FUNCTION_BLOCK L1_ControllerBase_SFC

VAR CONSTANT
	MAX_ERRORS	: UINT := 10;
	MAX_TIMEOUT	: TIME := T#30S;
END_VAR

VAR_INPUT
	dr			: REFERENCE TO L1_Director;		// acceso a todos los tiempos de espera
	IC			: BOOL;
	Execute		: BOOL;
	Ack			: BOOL;	
	SFCPause	: BOOL;
	SFCReset	: BOOL;
	UnsafeStop 	: BOOL := FALSE;
	Clocks		: ARRAY[1..MAX_ERRORS]	OF TON; 
END_VAR

VAR_OUTPUT
	Ready		: BOOL;
	Done		: BOOL := FALSE;
	Timed		: ARRAY[1..MAX_ERRORS]	OF BOOL; 
	NumError	: UINT := 0;
	gmModePrev	: L1_GEMMA := L1_GEMMA.A6Inicializando;
	
	colPicFill	: DWORD; // color para destacar en la foto según esté Ready (tranparente), Ejecutando (amarillo) o Esperando Ack (verde) 
	colPicFram	: DWORD; // color del marco  	
END_VAR

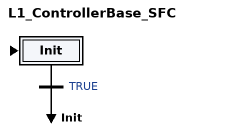
INITIAL_STEP Init:
END_STEP
TRANSITION FROM Init TO Init
    := TRUE;
END_TRANSITION

METHOD FB_init : BOOL
VAR_INPUT
	bInitRetains : BOOL; // if TRUE, the retain variables are initialized (warm start / cold start)
	bInCopyCode : BOOL;  // if TRUE, the instance afterwards gets moved into the copy code (online change)
END_VAR

VAR 
	I: UINT;
END_VAR
NumError		:= 0;					// Inicializar el estado a 0 (no hay error)

FOR I:=1 TO MAX_ERRORS DO				// Inicializar todos los flags de etapas temporizadas
	Timed[i] 		:= FALSE;
	//Clocks[i].IN	:= Timed[i];
	//Clocks[i].PT	:= MAX_TIMEOUT;	
END_FOR
END_METHOD

METHOD IsPaused : BOOL
IsPaused := SFCPause;
END_METHOD

METHOD ProcessCycle : BOOL

VAR_INPUT
	gmMode : L1_GEMMA;
END_VAR

VAR 
	i : UINT;
END_VAR
// Tratamiento del reset
IF gmModePrev<>gmMode AND gmMode=L1_GEMMA.A6Inicializando THEN
	gmModePrev	:= gmMode;
	SFCReset 	:= TRUE;
ELSE
	SFCReset 	:= FALSE;
END_IF
gmModePrev := gmMode;

// Tratamiento de la parada
SFCPause := NOT UnsafeStop AND (NumError <> 0 OR gmMode=L1_GEMMA.A3ParadaEstado OR gmMode=L1_GEMMA.A4ParadaObtenida);

// Tratamiento de errores
FOR i:= 1 TO MAX_ERRORS DO			
	Clocks[i](IN:= Timed[i], PT:=MAX_TIMEOUT);
	IF Clocks[i].Q THEN								// si saltó algún temporizador, devolver su número como error
		NumError := i;
		EXIT;
	END_IF
END_FOR


// Tratamiento del color en la foto
IF Ready THEN
	colPicFill	:= colModFillReady;
	colPicFram	:= colModFramReady;
ELSIF Done THEN 
	colPicFill	:= colModFillDone;
	colPicFram	:= colModFramDone;	
ELSE
	colPicFill	:= colModFillExec;
	colPicFram	:= colModFramExec;	
END_IF
END_METHOD

METHOD ResetError : BOOL
NumError := 0;
END_METHOD

END_FUNCTION_BLOCK

(* stored: Version 1.1.0.1, ProductVersion 3.1.4024.11
   POU L1_ControllerBase_SFC: Id {b4a568e5-b860-4b97-ba61-d1f48d9d8c8d}, SpecialFunc None
   Method FB_init: Id {0d874f96-f55f-4d86-871c-77c076024b66}
   Method IsPaused: Id {e98f7813-c900-4fd4-9a12-006983f9c884}
   Method ProcessCycle: Id {c358a4ee-9530-49d3-9f5f-b83d275d2af8}
   Method ResetError: Id {ca1cc05a-c1aa-4e32-b999-d986fdd3d9f7} *)
